{attribute 'qualified_only'}
VAR_GLOBAL
		EC : EC_245FBB9A;
END_VAR

(* stored: Version 1.2.0.0
   GVL GVL_iXlinker: Id {4cabe4e6-6ccc-4b92-b0d0-c1d5db34e8f9} *)
